PROGRAM MAIN
VAR
	test AT %Q* : BYTE;
END_VAR

END_PROGRAM

(* stored: Version 1.1.0.1, ProductVersion 3.1.4024.11
   POU MAIN: Id {b13e881b-2fb2-49ff-a953-4bcb05c0b5ab}, SpecialFunc None *)
